(* IEC 61131-3 sources: POC_HINCAPIE/Project/SIEMENS/DIGSI/Guadalupe/TMP/CFC/7344242.1412 (part 2) *)

     (* 0137 - GDL69TRF2F002_.Application.FG1_UserDef.FB3_Universal.RxPosQ013.DPC_StatusOn *)
     EXV_SPS_0137   {COMMENT := "GDL69TRF2F002_.Application.FG1_UserDef.FB3_Universal.RxPosQ013.DPC_StatusOn";DESC := "0##Application#Usuario#Rx Goose#Posicion 9T6-Q0#closed##1";}:IEXV_SPS_BO;

     (* 0138 - GDL69TRF2F002_.Application.FG1_UserDef.FB3_Universal.Rx86BFB169 *)
     EXV_SPS_0138   {COMMENT := "GDL69TRF2F002_.Application.FG1_UserDef.FB3_Universal.Rx86BFB169";DESC := "0##Application#Usuario#Rx Goose#Opero 86BF B1 69 kV##1";}:IEXV_SPS_BO;

     (* 0139 - GDL69TRF2F002_.Application.FG1_UserDef.FB3_Universal.Rx86BFB269 *)
     EXV_SPS_0139   {COMMENT := "GDL69TRF2F002_.Application.FG1_UserDef.FB3_Universal.Rx86BFB269";DESC := "0##Application#Usuario#Rx Goose#Opero 86BF B2 69 kV##1";}:IEXV_SPS_BO;

     (* 0140 - GDL69TRF2F002_.Application.FG1_UserDef.FB3_Universal.Rx86BF13 *)
     EXV_SPS_0140   {COMMENT := "GDL69TRF2F002_.Application.FG1_UserDef.FB3_Universal.Rx86BF13";DESC := "0##Application#Usuario#Rx Goose#Opero 86BF 13.8 kV##1";}:IEXV_SPS_BO;

     (* 0141 - GDL69TRF2F002_.Application.FG1_UserDef.FB1_Universal.SPS1 *)
     EXV_SPS_0141   {COMMENT := "GDL69TRF2F002_.Application.FG1_UserDef.FB1_Universal.SPS1";DESC := "0##Application#Usuario#Entradas#Posicion Q1 Cerrado##1";}:IEXV_SPS_BO;

     (* 0142 - GDL69TRF2F002_.Application.FG1_UserDef.FB1_Universal.FaPTN2PCyMHV *)
     EXV_SPS_0142   {COMMENT := "GDL69TRF2F002_.Application.FG1_UserDef.FB1_Universal.FaPTN2PCyMHV";DESC := "0##Application#Usuario#Entradas#Falla MCB PT B1_2 69kV PCyM N2##1";}:IEXV_SPS_BO;

     (* 0143 - GDL69TRF2F002_.Application.FG1_UserDef.FB1_Universal.FaPTN2Bar1HV *)
     EXV_SPS_0143   {COMMENT := "GDL69TRF2F002_.Application.FG1_UserDef.FB1_Universal.FaPTN2Bar1HV";DESC := "0##Application#Usuario#Entradas#Falla MCB PT B1 69kV 6TUJ1 N2##1";}:IEXV_SPS_BO;

     (* 0144 - GDL69TRF2F002_.Application.FG1_UserDef.FB3_Universal.RxPosQ2.DPC_StatusOn *)
     EXV_SPS_0144   {COMMENT := "GDL69TRF2F002_.Application.FG1_UserDef.FB3_Universal.RxPosQ2.DPC_StatusOn";DESC := "0##Application#Usuario#Rx Goose#Posicion 6T4-Q2#closed##1";}:IEXV_SPS_BO;

     (* 0145 - GDL69TRF2F002_.Application.FG1_UserDef.FB1_Universal.FaPTN2Bar2HV *)
     EXV_SPS_0145   {COMMENT := "GDL69TRF2F002_.Application.FG1_UserDef.FB1_Universal.FaPTN2Bar2HV";DESC := "0##Application#Usuario#Entradas#Falla MCB PT B2 69kV 6TUJ2 N2##1";}:IEXV_SPS_BO;

     (* 0146 - GDL69TRF2F002_.Application.FG1_UserDef.FB2_Universal.SPS *)
     EXV_SPS_0146   {COMMENT := "GDL69TRF2F002_.Application.FG1_UserDef.FB2_Universal.SPS";DESC := "0##Application#Usuario#Logicas#Condicion B1 OK##1";}:OEXV_BO_SPS;

     (* 0147 - GDL69TRF2F002_.Application.FG1_UserDef.FB2_Universal.SPS1 *)
     EXV_SPS_0147   {COMMENT := "GDL69TRF2F002_.Application.FG1_UserDef.FB2_Universal.SPS1";DESC := "0##Application#Usuario#Logicas#Condicion B2 OK##1";}:OEXV_BO_SPS;

     (* 0148 - GDL69TRF2F002_.Application.FG1_UserDef.FB2_Universal.SPS2 *)
     EXV_SPS_0148   {COMMENT := "GDL69TRF2F002_.Application.FG1_UserDef.FB2_Universal.SPS2";DESC := "0##Application#Usuario#Logicas#Condicion B1/B2 OK##1";}:OEXV_BO_SPS;
END_VAR

     EXV_SPS_0128        (LNK := 128);

     EXV_SPS_0129        (LNK := 129);

     EXV_SPS_0133        (LNK := 133);

     EXV_SPS_0134        (LNK := 134);

     EXV_SPS_0135        (LNK := 135);

     EXV_SPS_0136        (LNK := 136);

     EXV_SPS_0137        (LNK := 137);

     EXV_SPS_0138        (LNK := 138);

     EXV_SPS_0139        (LNK := 139);

     EXV_SPS_0140        (LNK := 140);

     EXV_SPS_0141        (LNK := 141);

     EXV_SPS_0142        (LNK := 142);

     EXV_SPS_0143        (LNK := 143);

     EXV_SPS_0144        (LNK := 144);

     EXV_SPS_0145        (LNK := 145);

     AND10_1             (X1 := EXV_SPS_0141.VAL(* POSITION := 29*5: SIZE := 31* -1:   *) ,
                          X2 := NOT EXV_SPS_0138.VAL(* POSITION := 29*6: SIZE := 31* -1:   *) ,
                          X3 := NOT EXV_SPS_0142.VAL(* POSITION := 23*7: SIZE := 37* -1:   *) ,
                          X4 := NOT EXV_SPS_0143.VAL(* POSITION := 24*8: SIZE := 36* -1:   *) ,
                          X5 := 1,
                          X6 := 1,
                          X7 := 1,
                          X8 := 1,
                          X9 := 1,
                          X10 := 1);

     AND10_2             (X1 := EXV_SPS_0144.VAL(* POSITION := 27*15: SIZE := 33* -1:   *) ,
                          X2 := NOT EXV_SPS_0139.VAL(* POSITION := 29*16: SIZE := 31* -1:   *) ,
                          X3 := NOT EXV_SPS_0142.VAL(* POSITION := 23*17: SIZE := 37* -1:   *) ,
                          X4 := NOT EXV_SPS_0145.VAL(* POSITION := 24*18: SIZE := 36* -1:   *) ,
                          X5 := 1,
                          X6 := 1,
                          X7 := 1,
                          X8 := 1,
                          X9 := 1,
                          X10 := 1);

     OR10_3              (X1 := AND10_1.Y,
                          X2 := AND10_2.Y,
                          X3 := 0,
                          X4 := 0,
                          X5 := 0,
                          X6 := 0,
                          X7 := 0,
                          X8 := 0,
                          X9 := 0,
                          X10 := 0);

     AND10_4             (X1 := OR10_3.Y,
                          X2 := NOT EXV_SPS_0135.VAL(* POSITION := 27*30: SIZE := 33* -1:   *) ,
                          X3 := NOT EXV_SPS_0137.VAL(* POSITION := 27*31: SIZE := 33* -1:   *) ,
                          X4 := NOT EXV_SPS_0136.VAL(* POSITION := 34*32: SIZE := 26* -1:   *) ,
                          X5 := NOT EXV_SPS_0140.VAL(* POSITION := 29*33: SIZE := 31* -1:   *) ,
                          X6 := 1,
                          X7 := 1,
                          X8 := 1,
                          X9 := 1,
                          X10 := 1);

     AND10_5             (X1 := NOT EXV_SPS_0133.VAL(* POSITION := 33*41: SIZE := 26* -1:   *) ,
                          X2 := NOT EXV_SPS_0128.VAL(* POSITION := 23*42: SIZE := 38* -1:   *) ,
                          X3 := EXV_SPS_0134.VAL(* POSITION := -1*-1: SIZE := 31* -1:   *) ,
                          X4 := EXV_SPS_0129.VAL(* POSITION := -1*-1: SIZE := 33* -1:   *) ,
                          X5 := 1,
                          X6 := 1,
                          X7 := 1,
                          X8 := 1,
                          X9 := 1,
                          X10 := 1);

     AND10_6             (X1 := AND10_4.Y,
                          X2 := AND10_5.Y,
                          X3 := 1,
                          X4 := 1,
                          X5 := 1,
                          X6 := 1,
                          X7 := 1,
                          X8 := 1,
                          X9 := 1,
                          X10 := 1);

     EXV_SPS_0130        (LNK := 130,
                          VAL := AND10_6.Y(* POSITION := 111*35: SIZE := 39* -1:   *) );
     EXV_SPS_0131        (LNK := 131,
                          VAL := AND10_4.Y(* POSITION := 83*24: SIZE := 34* -1:   *) );
     EXV_SPS_0132        (LNK := 132,
                          VAL := AND10_5.Y(* POSITION := 86*41: SIZE := 34* -1:   *) );
     EXV_SPS_0146        (LNK := 146,
                          VAL := AND10_1.Y(* POSITION := 88*5: SIZE := 29* -1:   *) );
     EXV_SPS_0147        (LNK := 147,
                          VAL := AND10_2.Y(* POSITION := 87*15: SIZE := 29* -1:   *) );
     EXV_SPS_0148        (LNK := 148,
                          VAL := OR10_3.Y(* POSITION := 107*9: SIZE := 30* -1:   *) );

(* COMMENT_TEXT;{X=3,Y=6};{Width=18, Height=1};FontSize := 8,LineColor := 0,LineWidth := 0,Alignment := Near,AutoWrap := True,BackColor := -256,Background := False,TextColor := 0,WallpaperGamma := 100,PartitionID := 1,;GOOSE 86BF B1 69kV No Op BCU *)
(* COMMENT_TEXT;{X=6,Y=31};{Width=14, Height=1};FontSize := 8,LineColor := 0,LineWidth := 0,Alignment := Near,AutoWrap := True,BackColor := -256,Background := False,TextColor := 0,WallpaperGamma := 100,PartitionID := 1,;GOOSE Pos 9T6-Q0 F004 *)
(* COMMENT_TEXT;{X=6,Y=33};{Width=19, Height=1};FontSize := 8,LineColor := 0,LineWidth := 0,Alignment := Near,AutoWrap := True,BackColor := -256,Background := False,TextColor := 0,WallpaperGamma := 100,PartitionID := 1,;GOOSE 86BF 13.8kV No Op F004 *)
(* COMMENT_TEXT;{X=3,Y=16};{Width=18, Height=1};FontSize := 8,LineColor := 0,LineWidth := 0,Alignment := Near,AutoWrap := True,BackColor := -256,Background := False,TextColor := 0,WallpaperGamma := 100,PartitionID := 1,;GOOSE 86BF B2 69kV No Op BCU *)
(* COMMENT_TEXT;{X=3,Y=15};{Width=18, Height=1};FontSize := 8,LineColor := 0,LineWidth := 0,Alignment := Near,AutoWrap := True,BackColor := -256,Background := False,TextColor := 0,WallpaperGamma := 100,PartitionID := 1,;GOOSE Pos Q2 F003 *)

END_PROGRAM

                                                  (* ---------- Program : CHART_Posiciones ----------  *)

PROGRAM CHART_Posiciones
{COMMENT := "Posiciones";DESC := "";}
(* ChartLayout;PageSize := A4,Rows := 3,Columns := 2,MarginMode := WithoutMargins,MarginSize := 37,MarginLines := 1 *)
(* PartitionInfo;Id := 1,Name := Partition_1,Comment :=   *)
VAR

     (* IO_IOVISIBILITY;OR10_1;X3:X4:X5:X6:X7:X8:X9:X10: *)

     (* PartitionInfo;PartitionID OR10_1;1  *)
OR10_1          { COMMENT := 'or10_5'; POSITION := 69,3; SIZE := 12, 12; } :OR10;

     (* IO_IOVISIBILITY;OR10_2;X3:X4:X5:X6:X7:X8:X9:X10: *)

     (* PartitionInfo;PartitionID OR10_2;1  *)
OR10_2          { COMMENT := 'or10_6'; POSITION := 69,10; SIZE := 12, 12; } :OR10;

     (* PartitionInfo;PartitionID BUILD_DPS_3;1  *)
BUILD_DPS_3     { COMMENT := 'build_dps_5'; POSITION := 92,3; SIZE := 12, 12; } :BUILD_DPS;

     (* PartitionInfo;PartitionID BUILD_DPS_4;1  *)
BUILD_DPS_4     { COMMENT := 'build_dps_1'; POSITION := 92,17; SIZE := 12, 12; } :BUILD_DPS;

     (* 0149 - GDL69TRF2F002_.Application.FG1_Breaker_3pol.FB1_XCBR.Pos *)
     EXV_DPS_0149   {COMMENT := "GDL69TRF2F002_.Application.FG1_Breaker_3pol.FB1_XCBR.Pos";DESC := "0##Application#Interruptor HV#Circuit break.#Position##1";}:OEXV_DS_DPS;

     (* 0150 - GDL69TRF2F002_.Application.FG2_Breaker_3pol.FB1_XCBR.Pos *)
     EXV_DPS_0150   {COMMENT := "GDL69TRF2F002_.Application.FG2_Breaker_3pol.FB1_XCBR.Pos";DESC := "0##Application#Interruptor LV#Circuit break.#Position##1";}:OEXV_DS_DPS;

     (* 0151 - GDL69TRF2F002_.Application.FG1_UserDef.FB1_Universal.SPS2 *)
     EXV_SPS_0151   {COMMENT := "GDL69TRF2F002_.Application.FG1_UserDef.FB1_Universal.SPS2";DESC := "0##Application#Usuario#Entradas#Posicion Int Q0 Cerrado##1";}:IEXV_SPS_BO;

     (* 0152 - GDL69TRF2F002_.Application.FG1_UserDef.FB3_Universal.RxPosQ069.DPC_StatusOn *)
     EXV_SPS_0152   {COMMENT := "GDL69TRF2F002_.Application.FG1_UserDef.FB3_Universal.RxPosQ069.DPC_StatusOn";DESC := "0##Application#Usuario#Rx Goose#Posicion 6T4-Q0#closed##1";}:IEXV_SPS_BO;

     (* 0153 - GDL69TRF2F002_.Application.FG1_UserDef.FB3_Universal.RxPosQ069.DPC_StatusOff *)
     EXV_SPS_0153   {COMMENT := "GDL69TRF2F002_.Application.FG1_UserDef.FB3_Universal.RxPosQ069.DPC_StatusOff";DESC := "0##Application#Usuario#Rx Goose#Posicion 6T4-Q0#open##1";}:IEXV_SPS_BO;

     (* 0154 - GDL69TRF2F002_.Application.FG1_UserDef.FB3_Universal.RxPosQ013.DPC_StatusOn *)
     EXV_SPS_0154   {COMMENT := "GDL69TRF2F002_.Application.FG1_UserDef.FB3_Universal.RxPosQ013.DPC_StatusOn";DESC := "0##Application#Usuario#Rx Goose#Posicion 9T6-Q0#closed##1";}:IEXV_SPS_BO;

     DEF_BUILD_DPS_3_QL:QUAL;

     DEF_BUILD_DPS_4_QL:QUAL;

END_VAR

DEF_BUILD_DPS_3_QL.VAL := 16#0000;
DEF_BUILD_DPS_4_QL.VAL := 16#0000;
     EXV_SPS_0151        (LNK := 151);

     EXV_SPS_0152        (LNK := 152);

     EXV_SPS_0153        (LNK := 153);

     EXV_SPS_0154        (LNK := 154);

     OR10_1              (X1 := EXV_SPS_0152.VAL(* POSITION := 29*6: SIZE := 33* -1:   *) ,
                          X2 := EXV_SPS_0151.VAL(* POSITION := 29*7: SIZE := 33* -1:   *) ,
                          X3 := 0,
                          X4 := 0,
                          X5 := 0,
                          X6 := 0,
                          X7 := 0,
                          X8 := 0,
                          X9 := 0,
                          X10 := 0);

     OR10_2              (X1 := NOT EXV_SPS_0151.VAL(* POSITION := 29*13: SIZE := 33* -1:   *) ,
                          X2 := EXV_SPS_0153.VAL(* POSITION := 30*14: SIZE := 32* -1:   *) ,
                          X3 := 0,
                          X4 := 0,
                          X5 := 0,
                          X6 := 0,
                          X7 := 0,
                          X8 := 0,
                          X9 := 0,
                          X10 := 0);

     BUILD_DPS_3         (IS_ON := OR10_1.Y,
                          IS_OFF := OR10_2.Y,
                          BAD_00 := 0,
                          QL := DEF_BUILD_DPS_3_QL);

     BUILD_DPS_4         (IS_ON := EXV_SPS_0154.VAL(* POSITION := -1*-1: SIZE := 33* -1:   *) ,
                          IS_OFF := NOT EXV_SPS_0154.VAL(* POSITION := -1*-1: SIZE := 33* -1:   *) ,
                          BAD_00 := 0,
                          QL := DEF_BUILD_DPS_4_QL);

     EXV_DPS_0149        (LNK := 149,
                          VAL := BUILD_DPS_3.OUT(* POSITION := 115*6: SIZE := 32* -1:   *) );
     EXV_DPS_0150        (LNK := 150,
                          VAL := BUILD_DPS_4.OUT(* POSITION := 115*20: SIZE := 32* -1:   *) );

(* COMMENT_TEXT;{X=4,Y=6};{Width=17, Height=1};FontSize := 10,LineColor := 0,LineWidth := 0,Alignment := Near,AutoWrap := True,BackColor := -256,Background := False,TextColor := 0,WallpaperGamma := 100,PartitionID := 1,;GOOSE Pos Q0 69kV BCU *)
(* COMMENT_TEXT;{X=4,Y=14};{Width=17, Height=1};FontSize := 10,LineColor := 0,LineWidth := 0,Alignment := Near,AutoWrap := True,BackColor := -256,Background := False,TextColor := 0,WallpaperGamma := 100,PartitionID := 1,;GOOSE Pos Q0 69kV BCU *)
(* COMMENT_TEXT;{X=4,Y=20};{Width=18, Height=1};FontSize := 10,LineColor := 0,LineWidth := 0,Alignment := Near,AutoWrap := True,BackColor := -256,Background := False,TextColor := 0,WallpaperGamma := 100,PartitionID := 1,;GOOSE Pos Q0 13.8kV F004 *)

END_PROGRAM

                                                  (* ---------- Program : CHART_Synchrocheck ----------  *)

PROGRAM CHART_Synchrocheck
{COMMENT := "Synchrocheck";DESC := "";}
(* ChartLayout;PageSize := A4,Rows := 3,Columns := 2,MarginMode := WithoutMargins,MarginSize := 37,MarginLines := 1 *)
(* PartitionInfo;Id := 1,Name := Partition_1,Comment :=    *)
VAR

     (* PartitionInfo;PartitionID DPC_DEF_1;1  *)
DPC_DEF_1       { COMMENT := 'dpc_def_1'; POSITION := 68,2; SIZE := 12, 12; } :DPC_DEF;

     (* PartitionInfo;PartitionID DPC_EXE_2;1  *)
DPC_EXE_2       { COMMENT := 'dpc_exe_1'; POSITION := 88,2; SIZE := 12, 12; } :DPC_EXE;

     (* 0155 - GDL69TRF2F002_.Application.FG1_Breaker_3pol.FB1_CSWI.Pos *)
     EXV_DPC_0155   {COMMENT := "GDL69TRF2F002_.Application.FG1_Breaker_3pol.FB1_CSWI.Pos";DESC := "0##Application#Interruptor HV#Control#Cmd. with feedback##1";}:IEXV_DPC_DC;

     (* 0156 - GDL69TRF2F002_.Application.FG1_UserDef.FB1_Universal.ClsManEmerg *)
     EXV_SPS_0156   {COMMENT := "GDL69TRF2F002_.Application.FG1_UserDef.FB1_Universal.ClsManEmerg";DESC := "0##Application#Usuario#Entradas#Cierre Manual Int Q0##1";}:IEXV_SPS_BO;
END_VAR

     EXV_DPC_0155        (ID_IN.IDX := 155);

     EXV_SPS_0156        (LNK := 156);

     DPC_DEF_1           (ID := EXV_DPC_0155.IDOUT(* POSITION := -1*-1: SIZE := 35* -1:   *) ,
                          EN_I := 1,
                          VAL := 1,
                          SELECT := 2,
                          OPERATE := 1,
                          TRIG := EXV_SPS_0156.VAL(* POSITION := -1*-1: SIZE := 32* -1:   *) ,
                          EDGE := 0,
                          ORIGIN := 5);

     DPC_EXE_2           (ID := DPC_DEF_1.ID_OUT,
                          EN_I := DPC_DEF_1.EN_O,
                          CANCEL := 0,
                          REL_EQ := 0,
                          REL_DBL := 0,
                          REL_PROT := 1,
                          REL_PLBY := 0,
                          REL_ILOC := 1,
                          RQ_SYNC := 1,
                          PT := 10);

END_PROGRAM

                                                  (* ---------- Program : CHART_Sincronismo ----------  *)

PROGRAM CHART_Sincronismo
{COMMENT := "Sincronismo";DESC := "";}
(* ChartLayout;PageSize := A4,Rows := 3,Columns := 2,MarginMode := WithoutMargins,MarginSize := 24,MarginLines := 1 *)
(* PartitionInfo;Id := 1,Name := Partition_1,Comment :=   *)
VAR

     (* PartitionInfo;PartitionID GT_D_1;1  *)
GT_D_1          { COMMENT := 'gt_d_1'; POSITION := 53,33; SIZE := 12, 12; } :GT_D;

     (* PartitionInfo;PartitionID GT_D_2;1  *)
GT_D_2          { COMMENT := 'gt_d_2'; POSITION := 53,39; SIZE := 12, 12; } :GT_D;

     (* PartitionInfo;PartitionID GT_D_3;1  *)
GT_D_3          { COMMENT := 'gt_d_3'; POSITION := 53,45; SIZE := 12, 12; } :GT_D;

     (* PartitionInfo;PartitionID LT_D_4;1  *)
LT_D_4          { COMMENT := 'lt_d_1'; POSITION := 53,51; SIZE := 12, 12; } :LT_D;

     (* PartitionInfo;PartitionID LT_D_5;1  *)
LT_D_5          { COMMENT := 'lt_d_5'; POSITION := 53,57; SIZE := 12, 12; } :LT_D;

     (* PartitionInfo;PartitionID LT_D_6;1  *)
LT_D_6          { COMMENT := 'lt_d_6'; POSITION := 53,63; SIZE := 12, 12; } :LT_D;

     (* PartitionInfo;PartitionID LT_D_7;1  *)
LT_D_7          { COMMENT := 'lt_d_2'; POSITION := 53,7; SIZE := 12, 12; } :LT_D;

     (* PartitionInfo;PartitionID LT_D_8;1  *)
LT_D_8          { COMMENT := 'lt_d_3'; POSITION := 53,13; SIZE := 12, 12; } :LT_D;

     (* PartitionInfo;PartitionID LT_D_9;1  *)
LT_D_9          { COMMENT := 'lt_d_4'; POSITION := 53,19; SIZE := 12, 12; } :LT_D;

     (* IO_IOVISIBILITY;AND10_10;X7:X8:X9:X10: *)

     (* PartitionInfo;PartitionID AND10_10;1  *)
AND10_10        { COMMENT := 'and10_2'; POSITION := 89,46; SIZE := 12, 12; } :AND10;

     (* PartitionInfo;PartitionID LT_D_11;1  *)
LT_D_11         { COMMENT := 'lt_d_7'; POSITION := 195,32; SIZE := 12, 12; } :LT_D;

     (* IO_IOVISIBILITY;AND10_12;X4:X5:X6:X7:X8:X9:X10: *)

     (* PartitionInfo;PartitionID AND10_12;1  *)
AND10_12        { COMMENT := 'and10_1'; POSITION := 87,11; SIZE := 12, 12; } :AND10;

     (* IO_IOVISIBILITY;AND10_13;X3:X4:X5:X6:X7:X8:X9:X10: *)

     (* PartitionInfo;PartitionID AND10_13;1  *)
AND10_13        { COMMENT := 'and10_4'; POSITION := 213,11; SIZE := 12, 12; } :AND10;

     (* IO_IOVISIBILITY;AND10_14;X3:X4:X5:X6:X7:X8:X9:X10: *)

     (* PartitionInfo;PartitionID AND10_14;1  *)
AND10_14        { COMMENT := 'and10_3'; POSITION := 213,3; SIZE := 12, 12; } :AND10;

     (* IO_IOVISIBILITY;OR10_15;X3:X4:X5:X6:X7:X8:X9:X10: *)

     (* PartitionInfo;PartitionID OR10_15;1  *)
OR10_15         { COMMENT := 'or10_1'; POSITION := 243,19; SIZE := 12, 12; } :OR10;

     (* 0157 - GDL69TRF2F002_.Application.FG1_PowerTransformerSide.FN1_OMV_Fund_3ph.FB1_OpMeas_Fund_3ph_Pres.PhV.WYE_MV_PHSA_Mag *)
     EXV_MV_0157    {COMMENT := "GDL69TRF2F002_.Application.FG1_PowerTransformerSide.FN1_OMV_Fund_3ph.FB1_OpMeas_Fund_3ph_Pres.PhV.WYE_MV_PHSA_Mag";DESC := "0##Application#Transformador HV#Fund./sym.comp.#Fundam#Vph#phs A magn.##1";}:IEXV_MVL_DI;

     (* 0158 - GDL69TRF2F002_.Application.FG1_PowerTransformerSide.FN1_OMV_Fund_3ph.FB1_OpMeas_Fund_3ph_Pres.PhV.WYE_MV_PHSB_Mag *)
     EXV_MV_0158    {COMMENT := "GDL69TRF2F002_.Application.FG1_PowerTransformerSide.FN1_OMV_Fund_3ph.FB1_OpMeas_Fund_3ph_Pres.PhV.WYE_MV_PHSB_Mag";DESC := "0##Application#Transformador HV#Fund./sym.comp.#Fundam#Vph#phs B magn.##1";}:IEXV_MVL_DI;

     (* 0159 - GDL69TRF2F002_.Application.FG1_PowerTransformerSide.FN1_OMV_Fund_3ph.FB1_OpMeas_Fund_3ph_Pres.PhV.WYE_MV_PHSC_Mag *)
     EXV_MV_0159    {COMMENT := "GDL69TRF2F002_.Application.FG1_PowerTransformerSide.FN1_OMV_Fund_3ph.FB1_OpMeas_Fund_3ph_Pres.PhV.WYE_MV_PHSC_Mag";DESC := "0##Application#Transformador HV#Fund./sym.comp.#Fundam#Vph#phs C magn.##1";}:IEXV_MVL_DI;

     (* 0160 - GDL69TRF2F002_.Application.FG1_UserDef.FB2_Universal.SPS8 *)
     EXV_SPS_0160   {COMMENT := "GDL69TRF2F002_.Application.FG1_UserDef.FB2_Universal.SPS8";DESC := "0##Application#Usuario#Logicas#Barra Muerta##1";}:OEXV_BO_SPS;

     (* 0161 - GDL69TRF2F002_.Application.FG1_UserDef.FB2_Universal.SPS7 *)
     EXV_SPS_0161   {COMMENT := "GDL69TRF2F002_.Application.FG1_UserDef.FB2_Universal.SPS7";DESC := "0##Application#Usuario#Logicas#Barra Viva##1";}:OEXV_BO_SPS;

     (* 0162 - GDL69TRF2F002_.Application.FG1_UserDef.FB2_Universal.SPS9 *)
     EXV_SPS_0162   {COMMENT := "GDL69TRF2F002_.Application.FG1_UserDef.FB2_Universal.SPS9";DESC := "0##Application#Usuario#Logicas#13.8 kV Muerto##1";}:OEXV_BO_SPS;

     (* 0163 - GDL69TRF2F002_.Application.FG1_UserDef.FB2_Universal.SPS10 *)
     EXV_SPS_0163   {COMMENT := "GDL69TRF2F002_.Application.FG1_UserDef.FB2_Universal.SPS10";DESC := "0##Application#Usuario#Logicas#Condicion de Sincronismo##1";}:OEXV_BO_SPS;

     (* 0164 - GDL69TRF2F002_.Application.FG1_UserDef.FB2_Universal.SPS5 *)
     EXV_SPS_0164   {COMMENT := "GDL69TRF2F002_.Application.FG1_UserDef.FB2_Universal.SPS5";DESC := "0##Application#Usuario#Logicas#Barra Muerta - Linea muerta##1";}:OEXV_BO_SPS;

     (* 0165 - GDL69TRF2F002_.Application.FG1_UserDef.FB2_Universal.SPS6 *)
     EXV_SPS_0165   {COMMENT := "GDL69TRF2F002_.Application.FG1_UserDef.FB2_Universal.SPS6";DESC := "0##Application#Usuario#Logicas#Barra Viva - Linea muerta##1";}:OEXV_BO_SPS;

     (* 0166 - GDL69TRF2F002_.Application.FG1_PowerTransformerStarpoint.FN1_OMV_Fund_1ph.FB1_OpMeas_Fund_1ph_Pres.VxC.CMV_Mag *)
     EXV_MV_0166    {COMMENT := "GDL69TRF2F002_.Application.FG1_PowerTransformerStarpoint.FN1_OMV_Fund_1ph.FB1_OpMeas_Fund_1ph_Pres.VxC.CMV_Mag";DESC := "0##Application#Transform. neut.p 1#Fundamental#Fundam#V#magnitude##1";}:IEXV_MVL_DI;
END_VAR

     EXV_MV_0157         (LNK := 157);

     EXV_MV_0158         (LNK := 158);

     EXV_MV_0159         (LNK := 159);

     EXV_MV_0166         (LNK := 166);

     GT_D_1              (IN1 := EXV_MV_0157.VAL(* POSITION := -1*-1: SIZE := 41* -1:   *) ,
                          IN2 := 80);

     GT_D_2              (IN1 := EXV_MV_0158.VAL(* POSITION := -1*-1: SIZE := 41* -1:   *) ,
                          IN2 := 80);

     GT_D_3              (IN1 := EXV_MV_0159.VAL(* POSITION := -1*-1: SIZE := 41* -1:   *) ,
                          IN2 := 80);

     LT_D_4              (IN1 := EXV_MV_0157.VAL(* POSITION := -1*-1: SIZE := 41* -1:   *) ,
                          IN2 := 110);

     LT_D_5              (IN1 := EXV_MV_0158.VAL(* POSITION := -1*-1: SIZE := 41* -1:   *) ,
                          IN2 := 110);

     LT_D_6              (IN1 := EXV_MV_0159.VAL(* POSITION := -1*-1: SIZE := 41* -1:   *) ,
                          IN2 := 110);

     LT_D_7              (IN1 := EXV_MV_0157.VAL(* POSITION := -1*-1: SIZE := 41* -1:   *) ,
                          IN2 := 40);

     LT_D_8              (IN1 := EXV_MV_0158.VAL(* POSITION := -1*-1: SIZE := 41* -1:   *) ,
                          IN2 := 40);

     LT_D_9              (IN1 := EXV_MV_0159.VAL(* POSITION := -1*-1: SIZE := 41* -1:   *) ,
                          IN2 := 40);

     AND10_10            (X1 := GT_D_1.OUT,
                          X2 := GT_D_2.OUT,
                          X3 := GT_D_3.OUT,
                          X4 := LT_D_4.OUT,
                          X5 := LT_D_5.OUT,
                          X6 := LT_D_6.OUT,
                          X7 := 1,
                          X8 := 1,
                          X9 := 1,
                          X10 := 1);

     LT_D_11             (IN1 := EXV_MV_0166.VAL(* POSITION := -1*-1: SIZE := 38* -1:   *) ,
                          IN2 := 23);

     AND10_12            (X1 := LT_D_7.OUT,
                          X2 := LT_D_8.OUT,
                          X3 := LT_D_9.OUT,
                          X4 := 1,
                          X5 := 1,
                          X6 := 1,
                          X7 := 1,
                          X8 := 1,
                          X9 := 1,
                          X10 := 1);

     AND10_13            (X1 := AND10_10.Y,
                          X2 := LT_D_11.OUT,
                          X3 := 1,
                          X4 := 1,
                          X5 := 1,
                          X6 := 1,
                          X7 := 1,
                          X8 := 1,
                          X9 := 1,
                          X10 := 1);

     AND10_14            (X1 := AND10_12.Y,
                          X2 := LT_D_11.OUT,
                          X3 := 1,
                          X4 := 1,
                          X5 := 1,
                          X6 := 1,
                          X7 := 1,
                          X8 := 1,
                          X9 := 1,
                          X10 := 1);

     OR10_15             (X1 := 0,
                          X2 := AND10_13.Y,
                          X3 := 0,
                          X4 := 0,
                          X5 := 0,
                          X6 := 0,
                          X7 := 0,
                          X8 := 0,
                          X9 := 0,
                          X10 := 0);

     EXV_SPS_0160        (LNK := 160,
                          VAL := AND10_12.Y(* POSITION := -1*-1: SIZE := 27* -1:   *) );
     EXV_SPS_0161        (LNK := 161,
                          VAL := AND10_10.Y(* POSITION := -1*-1: SIZE := 26* -1:   *) );
     EXV_SPS_0162        (LNK := 162,
                          VAL := LT_D_11.OUT(* POSITION := -1*-1: SIZE := 28* -1:   *) );
     EXV_SPS_0163        (LNK := 163,
                          VAL := OR10_15.Y(* POSITION := -1*-1: SIZE := 33* -1:   *) );
     EXV_SPS_0164        (LNK := 164,
                          VAL := AND10_14.Y(* POSITION := -1*-1: SIZE := 35* -1:   *) );
     EXV_SPS_0165        (LNK := 165,
                          VAL := AND10_13.Y(* POSITION := -1*-1: SIZE := 34* -1:   *) );

(* COMMENT_TEXT;{X=65,Y=2};{Width=23, Height=3};FontSize := 10,LineColor := 0,LineWidth := 0,Alignment := Near,AutoWrap := True,BackColor := -16711681,Background := False,TextColor := 0,WallpaperGamma := 100,PartitionID := 1,;Condición de barra muerta *)
(* COMMENT_TEXT;{X=59,Y=28};{Width=22, Height=2};FontSize := 10,LineColor := 0,LineWidth := 0,Alignment := Near,AutoWrap := True,BackColor := -16711681,Background := False,TextColor := 0,WallpaperGamma := 100,PartitionID := 1,;Condición de barra viva *)
(* COMMENT_TEXT;{X=182,Y=26};{Width=22, Height=2};FontSize := 10,LineColor := 0,LineWidth := 0,Alignment := Near,AutoWrap := True,BackColor := -16711681,Background := False,TextColor := 0,WallpaperGamma := 100,PartitionID := 1,;Lado 13,8 KV Muerto *)

END_PROGRAM

CONFIGURATION  PLC_CONTROL
   RESOURCE PLANS { COMMENT := "Txt100_100";} ON CPU32
     TASK EVENT_SLOW     { TICKS := 1300;}(PRIORITY := INTERNAL);
     TASK EVENT_FAST     { TICKS := 255;}(PRIORITY := INTERNAL);
     TASK MEASUREMENT    { TICKS := 2536;}(PRIORITY := INTERNAL);
     TASK INTERLOCKING   { TICKS := 2173;}(PRIORITY := INTERNAL);

     PROGRAM FBI001 WITH EVENT_SLOW:  CHART_Alarmas;
     PROGRAM FBI002 WITH EVENT_FAST:  CHART_Arranque_50BF;
     PROGRAM FBI003 WITH EVENT_SLOW:  CHART_Disparo_por_Fases;
     PROGRAM FBI004 WITH EVENT_SLOW:  CHART_Falla_Goose;
     PROGRAM FBI005 WITH EVENT_SLOW:  CHART_Falla_PTs;
     PROGRAM FBI006 WITH EVENT_SLOW:  CHART_Interlocking;
     PROGRAM FBI007 WITH EVENT_SLOW:  CHART_Posiciones;
     PROGRAM FBI008 WITH EVENT_SLOW:  CHART_Synchrocheck;
     PROGRAM FBI009 WITH EVENT_SLOW:  CHART_Sincronismo;

   END_RESOURCE

 END_CONFIGURATION
